PROGRAM pouMsgMc
VAR
	
	
	
END_VAR

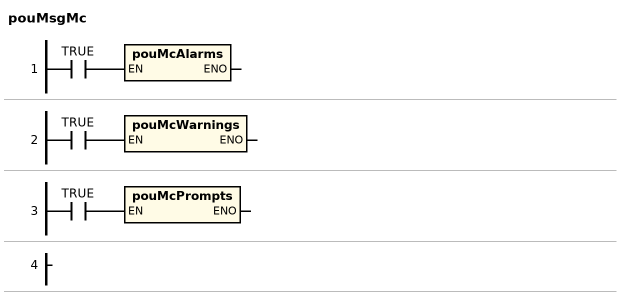
// NETWORK 1
pouMcAlarms();

// NETWORK 2
pouMcWarnings();

// NETWORK 3
pouMcPrompts();

// NETWORK 4

END_PROGRAM

(* stored: Version 1.1.0.1, ProductVersion 3.1.4024.12
   POU pouMsgMc: Id {5c98fced-520c-41b6-8a33-433000196d9d}, SpecialFunc None *)
